ABB RobotStudio station: Montaje_Herramienta.rsstnx

Station Montaje_Herramienta (saved by RobotStudio 23.4.10609.1)
Controller Controlador1
  mechanical unit ROB_1: IRB140_6_81_C_03, 6 joints, base frame (0, 0, 0) mm
Layout (positions relative to the parent item):
  - IRB140_6_81_C_03 [mechanism, from %ABB.RobotStudio.Models.IRB140%\IRB140_6_81_C_G_03.rslib] at (0, 0, 0) mm; joint values [0, 0, 0, 0, 0, 0] (rad or m)
  - Porta_Marcador [mechanism] at (515, 0, 712) mm, rotated rx 0 ry 90 rz 0 deg
      TCP Punta at (-90.51, 0, 137.01) mm, rotated rx 0 ry -45 rz 180 deg
      links: Support_RS
Attachment: Porta_Marcador is attached to IRB140_6_81_C_03 / Link6
Targets, tools, work objects and paths stored in the station, written as RAPID:
! task T_ROB1
MODULE CalibData
  PERS tooldata Punta:=[TRUE,[[64,64,143.009668],[0.853553391,0.146446609,-0.353553391,0.353553391]],[1,[0,0,1],[1,0,0,0],0,0,0]];
ENDMODULE

